// TIA Portal V19 export
ORGANIZATION_BLOCK "Main"   // OB1, LAD, ProgramCycle
TITLE = "Main Program Sweep (Cycle)"
{ S7_Optimized_Access := 'TRUE' }
// stored: SetENOAutomatically false
   VAR_INPUT
      Initial_Call : Bool;   // Initial call of this OB
      Remanence : Bool;   // =True, if remanent data are available
   END_VAR
   VAR_TEMP   // added for the SCL form of the ladder/FBD networks
      _w1 : Bool;
      _w2 : Bool;
   END_VAR
BEGIN

REGION Network 1
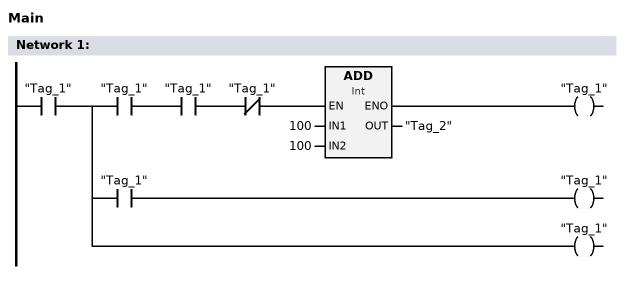
   RUNG wire#powerrail
      Contact( "Tag_1" )
      wire#w1
      Contact( "Tag_1" )
      Contact( "Tag_1" )
      I_Contact( "Tag_1" )
      { S7_Templates := "SrcType := Int" } Add(in1 := 100, in2 := 100, out => "Tag_2")
      Coil( "Tag_1" )
   END_RUNG
   RUNG wire#w1
      Contact( "Tag_1" )
      Coil( "Tag_1" )
   END_RUNG
   RUNG wire#w1
      Coil( "Tag_1" )
   END_RUNG
   // the same network as SCL:
   #_w1 := "Tag_1" AND "Tag_1" AND "Tag_1" AND NOT "Tag_1";
   IF #_w1 THEN "Tag_2" := 100 + 100; END_IF;
   #_w2 := "Tag_1";
   "Tag_1" := #_w1;
   "Tag_1" := #_w2 AND "Tag_1";
   "Tag_1" := #_w2;
END_REGION
END_ORGANIZATION_BLOCK
